FUNCTION_BLOCK FB_CalculateAI
VAR_INPUT
END_VAR
VAR_OUTPUT
END_VAR
VAR
	wMinRawIn		: WORD := 0;
	wMaxRawIn		: WORD := 32767;
	wRawIn			: WORD;
	wMinEngIn		: WORD;
	wMaxEngIn		: WORD;
	lrCalVal			: lreal;
	sDescription 	: STRING;
	lrRes			: LREAL;
	
END_VAR

lrRes := WORD_TO_LREAL(wRawIn)/WORD_TO_LREAL(wMaxRawIn);
lrCalVal:= word_to_lreal(wMaxEngIn) * lrRes;

PROPERTY CalVal : LREAL
GET
Calval := lrCalVal;
END_GET
SET
lrCalVal := Calval;
END_SET
END_PROPERTY

PROPERTY Description : STRING
SET
sDescription := Description;
END_SET
END_PROPERTY

PROPERTY MaxEngIn : WORD
SET
wMaxEngIn := MaxEngIn;
END_SET
END_PROPERTY

PROPERTY MinEngIn : WORD
SET
wMinEngIn := MinEngIn;
END_SET
END_PROPERTY

PROPERTY RawIn : WORD
SET
wRawIn := RawIn;
END_SET
END_PROPERTY

END_FUNCTION_BLOCK

(* stored: Version 1.1.0.1, ProductVersion 3.1.4024.11
   POU FB_CalculateAI: Id {a6c90192-70c6-4243-bf6d-396050117d59}, SpecialFunc None
   Property CalVal: Id {af397cf3-0928-4bff-b3eb-aeb49c8e1d11}
   Get Get: Id {85e151f0-1c31-4c13-97dc-9776e9cac336}
   Set Set: Id {a13171ca-7404-4b29-8916-65c34c48aba3}
   Property Description: Id {cbbbf50f-2b80-4046-b0e8-1c6bce65ff9f}
   Set Set: Id {c4e9289c-9ecc-4ff3-b11f-e6b2b98ce63d}
   Property MaxEngIn: Id {03467a06-4a26-4190-acd3-99669d2afc76}
   Set Set: Id {acdfb422-bc28-4ff2-9164-cae3fd2f8aaa}
   Property MinEngIn: Id {32fb28d8-0849-4619-977e-7cd9b48f6080}
   Set Set: Id {4445036d-d7dd-440c-9bfa-9232a153cbb9}
   Property RawIn: Id {d3a1ef51-bca2-4303-b3bb-c4468ab43115}
   Set Set: Id {ca413d67-ec75-49f6-b622-b5603270f4a9} *)
